FUNCTION_BLOCK Cylinder (* Template for an empty basic function block *)
  (* Standard: 61499-2 *)
  (* Version 1.0, 2019-04-25, Duc Do Tran, OFFIS e.V. *)
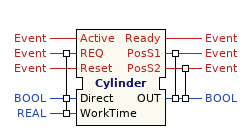
  EVENT_INPUT
    Active;
    REQ WITH Direct, WorkTime;
    Reset;
  END_EVENT
  EVENT_OUTPUT
    Ready;
    PosS1 WITH OUT;
    PosS2 WITH OUT;
  END_EVENT
  VAR_INPUT
    Direct : BOOL;
    WorkTime : REAL;
  END_VAR
  VAR_OUTPUT
    OUT : BOOL;
  END_VAR
  VAR
    GetTime : TIME; (* Internal Variable *)
    OldDirect : BOOL := 0; (* Internal Variable *)
  END_VAR
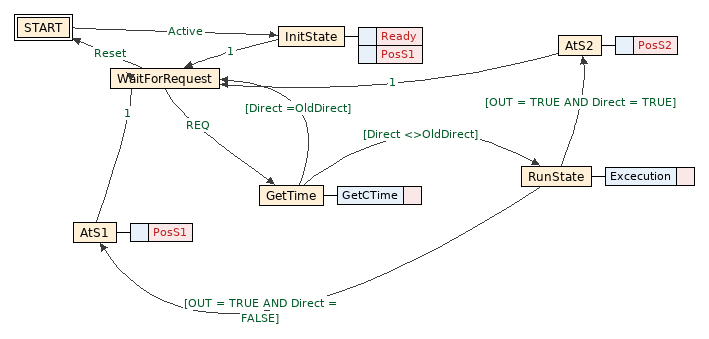
  EC_STATES
    START; (* Initial State *)
    AtS1 : -> PosS1;
    GetTime : GetCTime;
    RunState : Excecution;
    AtS2 : -> PosS2;
    InitState : -> Ready, -> PosS1;
    WaitForRequest;
  END_STATES
  EC_TRANSITIONS
    GetTime TO RunState := [Direct <>OldDirect];
    RunState TO AtS1 := [OUT = TRUE AND Direct = FALSE];
    RunState TO AtS2 := [OUT = TRUE AND Direct = TRUE];
    WaitForRequest TO GetTime := REQ;
    GetTime TO WaitForRequest := [Direct =OldDirect];
    START TO InitState := Active;
    InitState TO WaitForRequest := 1;
    AtS1 TO WaitForRequest := 1;
    AtS2 TO WaitForRequest := 1;
    WaitForRequest TO START := Reset;
  END_TRANSITIONS
  ALGORITHM Excecution IN ST: (* new algorithm *)
WHILE (TIME_IN_S_TO_LREAL(NOW_MONOTONIC() - GetTime) < WorkTime) DO
	OUT :=  FALSE;
END_WHILE;
OUT :=  TRUE;
OldDirect := Direct;
  END_ALGORITHM
  ALGORITHM GetCTime IN ST: (* new algorithm *)
GetTime := NOW_MONOTONIC();
  END_ALGORITHM
END_FUNCTION_BLOCK
